PROGRAM PRG_FB_CTRL_PID
VAR
	fSetpointValue					: LREAL		:= 5.0;
	fActualValue					: LREAL;
	fManSyncValue					: LREAL;
	bSync							: BOOL;

	fOut							: LREAL;
	bHold							: BOOL;

	eMode							: E_CTRL_MODE;
	stCTRL_PID_PARAMS				: ST_CTRL_PID_PARAMS;

	eErrorId						: E_CTRL_ERRORCODES;
	bError							: BOOL;
	bARWactive						: BOOL;

	(* controller *)
	fbCTRL_PID						: FB_CTRL_PID;

	bInit							: BOOL	:= TRUE;
	fbTON							: TON;
END_VAR

IF bInit THEN
	(* init parameter struct *)
	stCTRL_PID_PARAMS.tCtrlCycleTime		:= T#10ms;
	stCTRL_PID_PARAMS.tTaskCycleTime		:= T#10ms;
	stCTRL_PID_PARAMS.fKp					:= 20.0;			(* proportional gain Kp				*)
	stCTRL_PID_PARAMS.tTn					:= T#10S;		(*  Tn								*)
	stCTRL_PID_PARAMS.tTv					:= T#200MS;		(*  Tv								*)
	stCTRL_PID_PARAMS.tTd					:= T#100MS;		(*  Td								*)
	stCTRL_PID_PARAMS.fOutMaxLimit			:=  100;			(* maximum output limit				*)
	stCTRL_PID_PARAMS.fOutMinLimit			:= 0;			(* minimum output limit				*)

	(* set the mode to ACTIVE --> normal operation *)
	eMode := eCTRL_MODE_ACTIVE;

	(* reset the init flag *)
	bInit := FALSE;
END_IF


(* generate input signal *)
fbTON( IN:= TRUE,
		PT:= T#6S);
		
IF fbTON.Q THEN
	fbTON( IN:= FALSE);
	fSetpointValue := -1.0 * fSetpointValue;
END_IF

(* copy var to scope var *)
fSetpointValueToScope 	:= fSetpointValue;
fActualValueToScope 	:= fActualValue;


(* call controller *)
fbCTRL_PID(		fSetpointValue		:= fSetpointValue,
				fActualValue		:= fActualValue,
				fManSyncValue		:= fManSyncValue,
				bSync				:= bSync,
				eMode				:= eMode,
				bHold				:= bHold,
				stParams			:= stCTRL_PID_PARAMS,
				fOut				=> fOut,
				bARWactive			=> bARWactive,
				eErrorId			=> eErrorId,
				bError				=> bError
				);


(* copy var to scope var *)
fOutToScope := fOut;

END_PROGRAM

(* stored: Version 1.1.0.1
   POU PRG_FB_CTRL_PID: Id {ab4b9d68-903a-4dd7-8d89-3218bcdb26f1}, SpecialFunc None *)
